// Implicitly generated code : DO NOT EDIT
FUNCTION CheckRangeSigned : DINT
VAR_INPUT
	value, lower, upper: DINT;
END_VAR

// Implicitly generated code : Only an Implementation suggestion
{noflow}
IF (value < lower) THEN
	GVL_Checks.diCheckRangeSigned := GVL_Checks.diCheckRangeSigned +1;
	CheckRangeSigned := lower;
ELSIF(value > upper) THEN
	GVL_Checks.diCheckRangeSigned := GVL_Checks.diCheckRangeSigned +1;
	CheckRangeSigned := upper;
ELSE
	CheckRangeSigned := value;
END_IF
{flow}

END_FUNCTION

(* stored: Version 1.1.0.1, ProductVersion 3.1.4024.12
   POU CheckRangeSigned: Id {fa926bd1-bdc6-4409-a5cc-366b6901b2a5}, SpecialFunc CheckRangeSigned *)
